Fanuc KAREL source: ke00002.KL

-- PROVISIONAL review KL for V940-1; original PC SHA256 339f651a62ff188d03b329527c2411d3c8b4b735be9eb047bd0001f9504c8581
-- Incomplete behavior may be omitted. Consult companion uncertainty JSON. Do not deploy.
PROGRAM KE00002
%NOLOCKGROUP
BEGIN
  -- V9_ZERO_TABLE_METADATA_HINT layout=0002_ascii; no indexed target words; source/name/runtime held
  -- UNRESOLVED_PC offsets 5-17; opcodes 3F,75
  -- UNRESOLVED_PC offsets 22-29; opcodes 9D,23
  -- UNRESOLVED_PC offsets 34-46; opcodes 3F,22,9D,33,61
  -- UNRESOLVED_PC offsets 51-87; opcodes 27,22,2A,22,22,22,22,31
  -- UNRESOLVED_PC offsets 92-96; opcodes 7F
END KE00002
